Fanuc KAREL source: kt00021.KL

-- PROVISIONAL review KL for V940-1; original PC SHA256 c9e1b8253a12ccb947154aebac2d109d41e94b1abb0ea5093a6b9162ab2ef666
-- Incomplete behavior may be omitted. Consult companion uncertainty JSON. Do not deploy.
PROGRAM KT00021
%NOLOCKGROUP
VAR
  OUT : INTEGER
-- UNRESOLVED_DECL Y1 type=002018
-- UNRESOLVED_DECL Y2 type=002018
BEGIN
  -- V9_ZERO_TABLE_METADATA_HINT layout=0001; no indexed target words; source/name/runtime held
  -- UNRESOLVED_PC offsets 5-19; opcodes 2E,22,9D,33,B2
  -- UNRESOLVED_PC offsets 24-38; opcodes 2E,22,9D,33,B2
  -- UNRESOLVED_PC offsets 43-57; opcodes 2E,22,9D,33,B2
  -- UNRESOLVED_PC offsets 62-76; opcodes 2E,22,9D,33,B2
  -- UNRESOLVED_PC offsets 81-106; opcodes 22,9D,33,B1,22,9D,33,B1,52,23
  -- UNRESOLVED_PC offsets 111-115; opcodes 7F
END KT00021
